// TIA Portal project "Project4" (V15)

(* hardware
DEVICE "S7-1200 station_1"  S7-1200 Station
   slot 0: "Rack_0"  S7-1200 Rack  Rack  V1.0
   slot 1: "PLC_1"  CPU 1212C DC/DC/DC  6ES7 212-1AE40-0XB0  V4.2
*)

// ===== PLC "PLC_1"  CPU 1212C DC/DC/DC =====

VAR_GLOBAL   // PLC tag table "Default tag table"
   "Tag_1" AT %I0.6 : Bool;
   "Tag_2" AT %I0.7 : Bool;
   "Tag_3" AT %M0.5 : Bool;
   "Tag_4" AT %M0.1 : Bool;
   "Tag_5" AT %M0.0 : Bool;
   "Tag_6" AT %Q0.2 : Bool;
   "Tag_7" AT %Q0.3 : Bool;
   "Tag_8" AT %M0.3 : Bool;
   "Tag_9" AT %M1.1 : Bool;
END_VAR

ORGANIZATION_BLOCK "Main"   // OB1, LAD, ProgramCycle
TITLE = "Main Program Sweep (Cycle)"
{ S7_Optimized_Access := 'TRUE' }
VERSION : 0.1
   VAR_INPUT
      Initial_Call : Bool;   // Initial call of this OB
      Remanence : Bool;   // =True, if remanent data are available
   END_VAR
BEGIN

REGION Network 1
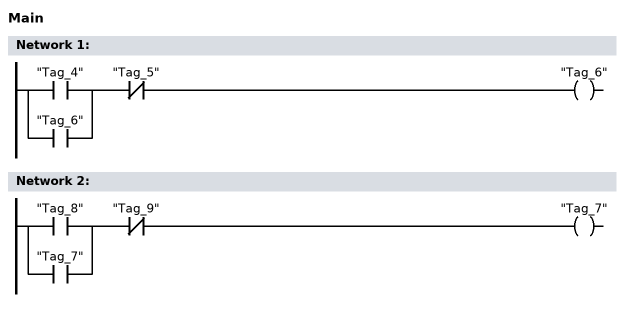
   RUNG wire#powerrail
      Contact( "Tag_4" )
      wire#w1
      I_Contact( "Tag_5" )
      Coil( "Tag_6" )
   END_RUNG
   RUNG wire#powerrail
      Contact( "Tag_6" )
   END_RUNG wire#w1
   // the same network as SCL:
   "Tag_6" := ("Tag_4" OR "Tag_6") AND NOT "Tag_5";
END_REGION

REGION Network 2
   RUNG wire#powerrail
      Contact( "Tag_8" )
      wire#w1
      I_Contact( "Tag_9" )
      Coil( "Tag_7" )
   END_RUNG
   RUNG wire#powerrail
      Contact( "Tag_7" )
   END_RUNG wire#w1
   // the same network as SCL:
   "Tag_7" := ("Tag_8" OR "Tag_7") AND NOT "Tag_9";
END_REGION
END_ORGANIZATION_BLOCK